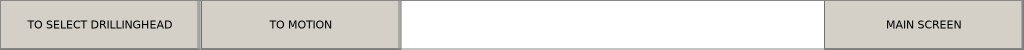
VISUALIZATION Nav  // 1024x50
    Button (0,0 200x50), "TO SELECT DRILLINGHEAD"
        OnMouseDown: change screen: SelectDrillinghead
    Button (201,0 200x50), "TO MOTION"
        OnMouseDown: change screen: Motion
    Button (824,0 200x50), "MAIN SCREEN"
        OnMouseDown: change screen: MainScreen
END_VISUALIZATION

(* stored: Version 1.1.0.1, ProductVersion 3.1.4024.12
   Visu Nav: Id {7421a2e2-aadb-4e59-af1a-edc393be95d1} *)
